INTERFACE I_ListItem EXTENDS __SYSTEM.IQueryInterface

END_INTERFACE

(* stored: Version 1.1.0.1, ProductVersion 3.1.4024.12
   Itf I_ListItem: Id {1fad1549-d200-406a-b21a-0c538dbe0c70} *)
